Staubli VAL3: moveBin.pgx

program moveBin()
begin
  movej(binPosition,flange,mFastMov)
  waitEndMove()
  message="moveBin:done"
  taskCreate "sendStatus",10,sendStatus()
  taskKill("moveBin")
end
